{attribute 'linkalways'} 
{attribute 'no_explicit_call' := 'This FB is a CLASS and must be accessed using methods or properties'}
{attribute 'enable_dynamic_creation'}
FUNCTION_BLOCK Node_F_VN_AddToContainerElements_DINT EXTENDS VisionNode
VAR
    nValue : _DINT(0);
    ipContainer : _ITcVnContainer;
    hrPrev : _HRESULT(S_OK);
    hresult : _HRESULT(S_OK);
END_VAR

METHOD PUBLIC  Clone : I_Node
VAR
    pNode : POINTER TO Node_F_VN_AddToContainerElements_DINT;
END_VAR
pNode := __NEW(Node_F_VN_AddToContainerElements_DINT);
Clone := pNode^;
END_METHOD

METHOD FB_init : BOOL
VAR_INPUT
    bInitRetains : BOOL; // if TRUE, the retain variables are initialized (warm start / cold start)
    bInCopyCode : BOOL;  // if TRUE, the instance afterwards gets moved into the copy code (online change)
END_VAR
AddParameter('nValue', nValue);
AddInput('ipContainer', ipContainer);
AddInput('hrPrev', hrPrev);
AddOutput('ipContainer', ipContainer);
AddOutput('hresult',hresult);
END_METHOD

METHOD PROTECTED OnExecute
hresult.Value := F_VN_AddToContainerElements_DINT(
    nValue := nValue.Value,
    ipContainer := ipContainer.Value,
    hrPrev:= hrPrev.Value);
END_METHOD

METHOD PUBLIC PreExecutionCheck
VAR_INPUT
    Check : I_PreExecutionChecks;
END_VAR
Check.IsTrue(ipContainer.IsValid, 'ipContainer must be a valid container');
Check.IsTrue(ipContainer.IsType(TC_GLOBAL_CONST_LIST.ContainerType_Vector_DINT), 'ipContainer contains incorrect type');
END_METHOD

END_FUNCTION_BLOCK

(* stored: Version 1.1.0.1, ProductVersion 3.1.4026.13
   POU Node_F_VN_AddToContainerElements_DINT: Id {3ca22ee4-32fb-4f73-bacc-f9740f95569f}, SpecialFunc None
   Folder Constructor: Id {35c20dd2-87cc-4566-86ba-fc5400c9f88b}
   Method Clone: Id {1a8b4e24-6256-4033-a451-346987bdc7f7}
   Method FB_init: Id {df9ad137-9e88-4adb-afb1-6c2542b80159}
   Method OnExecute: Id {6cbc37db-8738-4204-8b51-66e0719a4675}
   Method PreExecutionCheck: Id {03bdd54f-b150-434e-832b-bbf3da25d4f9} *)
